PROGRAM MAIN
VAR
END_VAR

Plc_Prog();

END_PROGRAM

(* stored: Version 1.1.0.1, ProductVersion 3.1.4024.9
   POU MAIN: Id {88845244-bcb1-4ed1-9462-4c7ef40b077e}, SpecialFunc None *)
